// TIA Portal project "colour_seperator_conveyor" (V18)
// Vorlageprojekt für das Buch mit Zielsystem S7-1200

(* hardware
DEVICE "S7-1200-Station_1"  S7-1200 Station
   slot 0: "Baugruppenträger_0"  Rack  V1.0
   slot 1: "PLC_1"  CPU 1211C DC/DC/DC  6ES7 211-1AE40-0XB0  V4.1
*)

// ===== PLC "PLC_1"  CPU 1211C DC/DC/DC =====

VAR_GLOBAL   // PLC tag table "Standard-Variablentabelle"
   "Tag_2" AT %E0.0 : Bool;
   "Tag_3" AT %E0.1 : Bool;
   "Tag_1" AT %A0.0 : Bool;
END_VAR

VAR_GLOBAL   // PLC tag table "OUTPUT_TAGS"
   "BELT_CONVEYOR_0" AT %Q0.1 : Bool;   // Ana Konveyör
   "PUSHER_0" AT %Q0.2 : Bool;   // Metalik renk iticisinin bobini
   "PUSHER_1" AT %Q0.3 : Bool;   // Yeşil renk iticisinin bobini
   "PUSHER_2" AT %Q0.4 : Bool;   // Mavi renk iticisinin bobini
   "BELT_CONVEYOR_1" AT %Q0.5 : Bool;   // Mavi renk konveyörü
   "BELT_CONVEYOR_2" AT %Q0.6 : Bool;   // Yeşil renk konveyörü
   "BELT_CONVEYOR_3" AT %Q0.7 : Bool;   // Metalik renk konveyörü
END_VAR

VAR_GLOBAL   // PLC tag table "INPUT_TAGS"
   "STOP" AT %I0.3 : Bool;   // STOP butonu
   "RETROREFLECTIVE_SENSOR_0" AT %I0.4 : Bool;   // Optik Sensör
   "PUSHER_0_BACKLIMIT" AT %I0.5 : Bool;   // Metalik renk iticisinin ileri reed sensörü
   "PUSHER_1_BACKLIMIT" AT %I0.6 : Bool;   // Yeşil renk iticisinin ileri reed sensörü
   "PUSHER_2_BACKLIMIT" AT %I0.7 : Bool;   // Mavi renk iticisinin ileri reed sensörü
   "DIFFUSE_SENSOR_0" AT %I1.0 : Bool;   // Mavi rnek konveyörün sınır sensörü
   "DIFFUSE_SENSOR_1" AT %I1.1 : Bool;   // Yeşil renk konveyörün sınır sensörü
   "DIFFUSE_SENSOR_2" AT %I1.2 : Bool;   // Metalik renk konveyörün sınır sensörü
   "VISION_SENSOR_0" AT %ID30 : DInt;   // Renk Sensörü (Mavi)
   "VISION_SENSOR_1" AT %ID34 : DInt;   // Renk Sensörü (Yeşil)
   "VISION_SENSOR_2" AT %ID38 : DInt;   // Renk Sensörü (Metalik)
END_VAR

DATA_BLOCK "data_block"   // DB1
{ S7_Optimized_Access := 'TRUE' }
VERSION : 0.1
BEGIN
END_DATA_BLOCK

// folder: System blocks/Program resources

DATA_BLOCK "IEC_Timer_0_DB"   // DB2
{ S7_Optimized_Access := 'TRUE' }
AUTHOR : Simatic
FAMILY : IEC
NAME : IEC_TMR
VERSION : 1.0
// stored: InstanceOfName IEC_TIMER
"IEC_TIMER"
BEGIN
END_DATA_BLOCK

DATA_BLOCK "TOF_DB"   // DB3
{ S7_Optimized_Access := 'TRUE' }
AUTHOR : Simatic
FAMILY : IEC
NAME : IEC_TMR
VERSION : 1.0
// stored: InstanceOfName IEC_TIMER
"IEC_TIMER"
BEGIN
END_DATA_BLOCK

DATA_BLOCK "IEC_Timer_0_DB_1"   // DB4
{ S7_Optimized_Access := 'TRUE' }
AUTHOR : Simatic
FAMILY : IEC
NAME : IEC_TMR
VERSION : 1.0
// stored: InstanceOfName IEC_TIMER
"IEC_TIMER"
BEGIN
END_DATA_BLOCK

DATA_BLOCK "IEC_Timer_0_DB_2"   // DB5
{ S7_Optimized_Access := 'TRUE' }
AUTHOR : Simatic
FAMILY : IEC
NAME : IEC_TMR
VERSION : 1.0
// stored: InstanceOfName IEC_TIMER
"IEC_TIMER"
BEGIN
END_DATA_BLOCK

// folder: (top level)

FUNCTION "Alternative_V1" : Void   // FC1, LAD
{ S7_Optimized_Access := 'TRUE' }
VERSION : 0.1
// RENK AYIRICI KONVEYÖR BANT PROJESİ
BEGIN

REGION Network 1: Ana Konveyör
   // Retroreflective sensörün çıkışı LOW olduğu zaman konveyör bant çalışmaya başlar. Konveyör bantın  
   // çalışma süresi motorun bantın başından sonuna kadar gitmek için harcadığı süredir. 10sn olarak 
   // tanımlanmıştır.
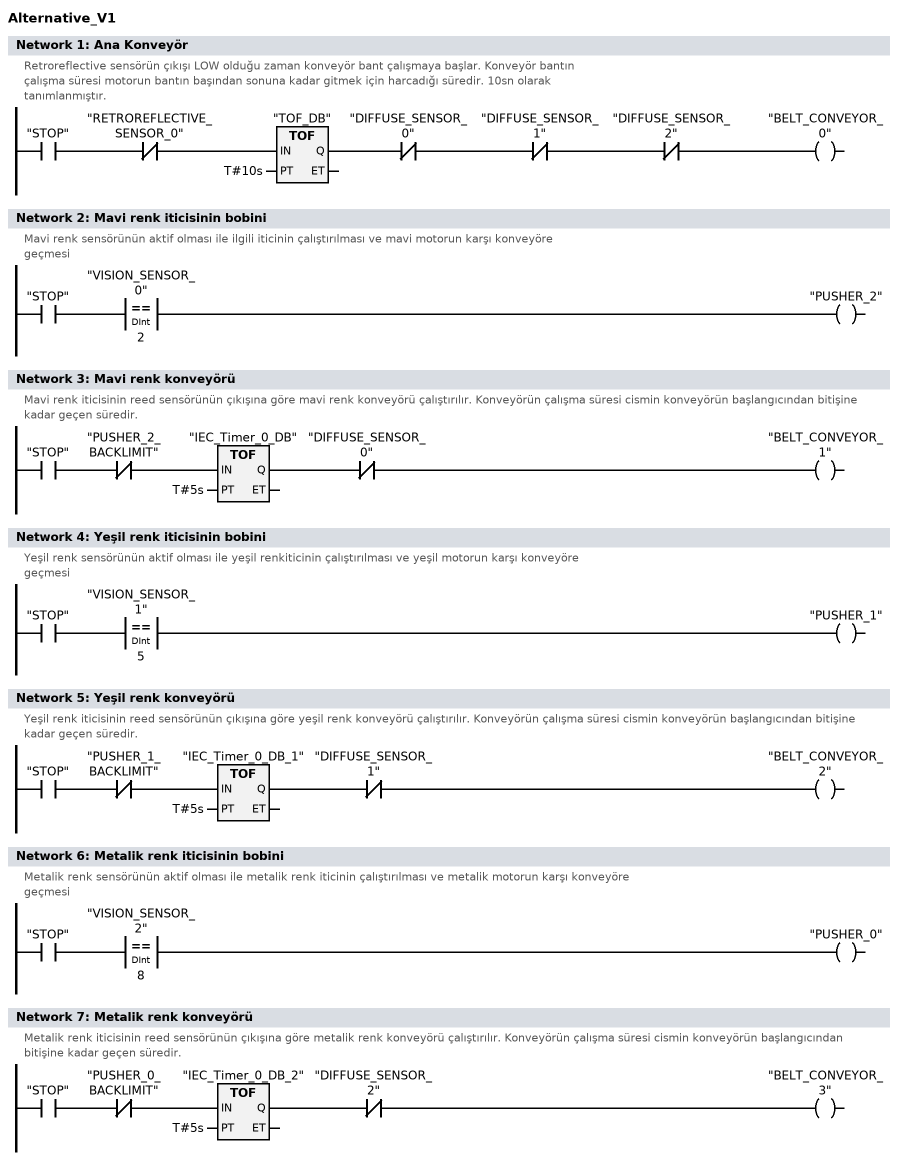
   "TOF_DB".TOF(IN := "STOP" AND NOT "RETROREFLECTIVE_SENSOR_0", PT := T#10s);
   "BELT_CONVEYOR_0" := "TOF_DB".Q AND NOT "DIFFUSE_SENSOR_0" AND NOT "DIFFUSE_SENSOR_1" AND NOT "DIFFUSE_SENSOR_2";
END_REGION

REGION Network 2: Mavi renk iticisinin bobini
   // Mavi renk sensörünün aktif olması ile ilgili iticinin çalıştırılması ve mavi motorun karşı konveyöre 
   // geçmesi
   RUNG wire#powerrail
      Contact( "STOP" )
      { S7_Templates := "SrcType := DInt" } EQ_Contact(in1 := "VISION_SENSOR_0", in2 := 2)
      Coil( "PUSHER_2" )
   END_RUNG
   // the same network as SCL:
   "PUSHER_2" := "STOP" AND ("VISION_SENSOR_0" = 2);
END_REGION

REGION Network 3: Mavi renk konveyörü
   // Mavi renk iticisinin reed sensörünün çıkışına göre mavi renk konveyörü çalıştırılır. Konveyörün çalışma süresi cismin konveyörün başlangıcından bitişine kadar geçen süredir.
   "IEC_Timer_0_DB".TOF(IN := "STOP" AND NOT "PUSHER_2_BACKLIMIT", PT := T#5s);
   "BELT_CONVEYOR_1" := "IEC_Timer_0_DB".Q AND NOT "DIFFUSE_SENSOR_0";
END_REGION

REGION Network 4: Yeşil renk iticisinin bobini
   // Yeşil renk sensörünün aktif olması ile yeşil renkiticinin çalıştırılması ve yeşil motorun karşı konveyöre 
   // geçmesi
   RUNG wire#powerrail
      Contact( "STOP" )
      { S7_Templates := "SrcType := DInt" } EQ_Contact(in1 := "VISION_SENSOR_1", in2 := 5)
      Coil( "PUSHER_1" )
   END_RUNG
   // the same network as SCL:
   "PUSHER_1" := "STOP" AND ("VISION_SENSOR_1" = 5);
END_REGION

REGION Network 5: Yeşil renk konveyörü
   // Yeşil renk iticisinin reed sensörünün çıkışına göre yeşil renk konveyörü çalıştırılır. Konveyörün çalışma süresi cismin konveyörün başlangıcından bitişine kadar geçen süredir.
   "IEC_Timer_0_DB_1".TOF(IN := "STOP" AND NOT "PUSHER_1_BACKLIMIT", PT := T#5s);
   "BELT_CONVEYOR_2" := "IEC_Timer_0_DB_1".Q AND NOT "DIFFUSE_SENSOR_1";
END_REGION

REGION Network 6: Metalik renk iticisinin bobini
   // Metalik renk sensörünün aktif olması ile metalik renk iticinin çalıştırılması ve metalik motorun karşı konveyöre 
   // geçmesi
   RUNG wire#powerrail
      Contact( "STOP" )
      { S7_Templates := "SrcType := DInt" } EQ_Contact(in1 := "VISION_SENSOR_2", in2 := 8)
      Coil( "PUSHER_0" )
   END_RUNG
   // the same network as SCL:
   "PUSHER_0" := "STOP" AND ("VISION_SENSOR_2" = 8);
END_REGION

REGION Network 7: Metalik renk konveyörü
   // Metalik renk iticisinin reed sensörünün çıkışına göre metalik renk konveyörü çalıştırılır. Konveyörün çalışma süresi cismin konveyörün başlangıcından bitişine kadar geçen süredir.
   "IEC_Timer_0_DB_2".TOF(IN := "STOP" AND NOT "PUSHER_0_BACKLIMIT", PT := T#5s);
   "BELT_CONVEYOR_3" := "IEC_Timer_0_DB_2".Q AND NOT "DIFFUSE_SENSOR_2";
END_REGION
END_FUNCTION

FUNCTION "MHJ-PLC-Lab-Function-S71200" : Void   // FC9000, SCL
{ S7_Optimized_Access := 'TRUE' }
VERSION : 0.1
   VAR_TEMP
      rdTimeReturn : Int;
      outputTime : DTL;
      SyncVal : Byte;
      forVal : Int;
      forVal_2 : Int;
      Value : Byte;
   END_VAR
   VAR CONSTANT
      CompVal : Byte := 16#34;
      Value_01 : Byte := 16#11;
      Value_01_DW : DWord := 16#A165_D992;
      Value_02_DW : DWord := 16#58BE_4401;
   END_VAR
BEGIN

   #Value:=PEEK(area := 16#82,
        dbNumber := 0,
        byteOffset := 511);
   #Value := #Value + 1;

   POKE(area := 16#82,
        dbNumber := 0,
        byteOffset := 511,
        value := #Value);

   POKE(area:=16#81,
        dbNumber:=0,
        byteOffset:=1016,
        value:=#Value_01_DW);
   POKE(area := 16#81,
        dbNumber := 0,
        byteOffset := 1020,
        value := #Value_02_DW);

   POKE(area := 16#81,
        dbNumber := 0,
        byteOffset := 511,
        value := B#16#00);

   FOR #forVal := 0 TO 120 DO
       FOR #forVal_2:=0 TO 10 DO
           #rdTimeReturn:=RD_SYS_T(#outputTime);
           #rdTimeReturn := WR_SYS_T(#outputTime);
           #rdTimeReturn := RD_SYS_T(#outputTime);
           #rdTimeReturn := WR_SYS_T(#outputTime);
       END_FOR;
       #SyncVal:= PEEK(area := 16#81,
                      dbNumber := 0,
                      byteOffset := 511);
       IF #SyncVal = #CompVal THEN
          GOTO M_1;
       END_IF;
   END_FOR;
   RETURN;

   M_1:
   POKE(area := 16#81,
        dbNumber := 0,
        byteOffset := 511,
        value := B#16#0);
END_FUNCTION

ORGANIZATION_BLOCK "Main"   // OB1, LAD, ProgramCycle
TITLE = "Main Program Sweep (Cycle)"
{ S7_Optimized_Access := 'TRUE' }
VERSION : 0.1
   VAR_INPUT
      Initial_Call : Bool;   // Initial call of this OB
      Remanence : Bool;   // =True, if remanent data are available
   END_VAR
BEGIN

REGION Network 1: Konnektierungsbaustein für PLC-Lab
   // Im Netzwerk 1 wird der Konnektierungsbaustein für PLC-Lab aufgerufen.
   // Dieser Aufruf darf nicht entfernt werden!
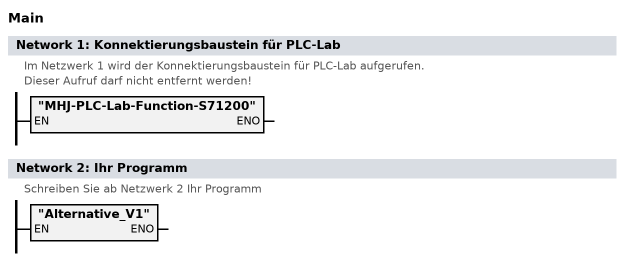
   RUNG wire#powerrail
      "MHJ-PLC-Lab-Function-S71200"()
   END_RUNG
   // the same network as SCL:
   "MHJ-PLC-Lab-Function-S71200"();
END_REGION

REGION Network 2: Ihr Programm
   // Schreiben Sie ab Netzwerk 2 Ihr Programm
   RUNG wire#powerrail
      "Alternative_V1"()
   END_RUNG
   // the same network as SCL:
   "Alternative_V1"();
END_REGION
END_ORGANIZATION_BLOCK